Yaskawa INFORM job: pipe_head_planes_program.JBI

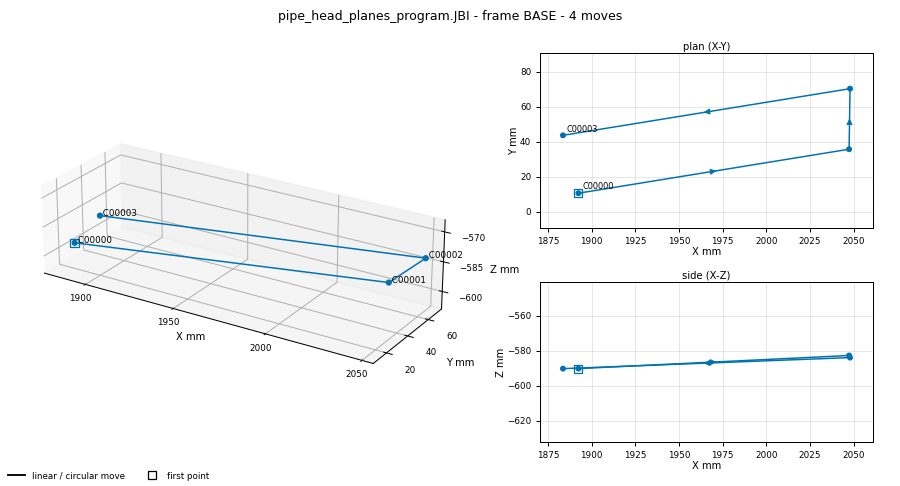
[picture p0: tool path of pipe_head_planes_program.JBI in frame BASE, 4 of 6 moves have a stored position in this frame; points joined in program order, loops and branches not executed]
/JOB
//NAME pipe_head_planes_program
//POS
///NPOS 4,0,4,0,0,0
///TOOL 0
///POSTYPE BASE
///RECTAN
///RCONF 0,0,0,0,0,0,0,0,0,0,0,0,0,0,0,0,0,0,0,0,0,0,0,0
C00000=1892.448407,10.612745,-590.213434,-175.000000,-5.000000,-5.000000
C00001=2047.403487,35.798664,-582.732018,-175.000000,-5.000000,-5.000000
C00002=2047.942711,70.453177,-583.927105,-175.000000,-5.000000,-5.000000
C00003=1883.603308,43.750182,-590.254390,-175.000000,-5.000000,-5.000000
///POSTYPE PULSE
///PULSE
EC00000=285696.0
EC00001=285696.0
EC00002=285696.0
EC00003=285696.0
//INST
///DATE 2023/08/13 11:14
///ATTR SC,RW,RJ
////FRAME BASE
///GROUP1 RB1,ST1
NOP
MOVJ P009 EX000 VJ=15.00
MOVJ C00000 EC00000 VJ=15.0
CALL JOB:SPYON
MOVL C00001 EC00001 V=150.0
MOVL C00002 EC00002 V=150.0
MOVL C00003 EC00003 V=150.0
CALL JOB:SPYOF
MOVJ P009 VJ=15.00
END
